PROGRAM Sorting
VAR
	
	Timerdelay0 : TON;
	Statustimer0 : BOOL;
	Timerdelay1 : TON;
	Statustimer1 : BOOL;
	Timerdelay2 : TON;
	Statustimer2 : BOOL;
	Timerdelay3 : TON;
	Statustimer3 : BOOL;
END_VAR

Timerdelay0(PT:=  T#5000MS , Q =>Statustimer0);
Timerdelay1(PT:=  T#1000MS , Q =>Statustimer1);
Timerdelay2(PT:=  T#1000MS , Q =>Statustimer2);
Timerdelay3(PT:=  T#800MS , Q =>Statustimer3);

(*
Do not turn conveyor on when GVL.X2_I3 slide is full 

IF GVL.X2_I0 THEN
	GVL.X2_00 := TRUE;
	END_IF
	IF Statustimer0 THEN
		GVL.X2_00 := FALSE;
	END_IF
	


Metallic workpiece (X2_I1) Wait and turn conveyor on then
 turn slide 1. 



*)

END_PROGRAM

(* stored: Version 1.1.0.1, ProductVersion 3.1.4024.15
   POU Sorting: Id {23aef86d-bd25-42f9-9306-f5a306b038a0}, SpecialFunc None *)
